Staubli VAL3: robotPut.pgx

public program robotPut(point pPosition, trsf trTrans, tool tTool, mdesc mApproach, mdesc mTarget)
  local point pAppro
begin
  // Places a part
  //
  // copyright (c) 2015 victortorreslopez
  //
  // GNU General Public License
  //
  // Parmeters
  // - pPosition: target position
  // - trTrans: approach transform to target position
  // - tTool: tool
  // - mApproach: movement descriptor to "approach" point
  // - mTarget: movement descriptor to "target" position
  //
  // Local variables
  // - pAppro: approach point to target position
  //
  // References
  // - "2005-27 Example Application". Staubli. 2005
  //
  // Version history
  // ---------------
  // 2.0, 2020/02/15, VTL: renames all parameters
  // 1.1, 2018/09/27, VTL: add "ma"
  // 1.0, 2018/09/27, VTL: rename "m" by "mt"
  // 0.0, 2015/01/14, VTL: alfa release
  //
  pAppro = appro(pPosition, trTrans)
  movej(pAppro, tTool, mApproach)
  movel(pPosition, tTool, mTarget)
  open(tTool)
  movel(pAppro, tTool, mTarget)
end
